FUNCTION_BLOCK E_CYCLE (* Peroidic event generator *)
  (* Standard: 61499-1 Annex A; Description: Copyright (c) 2017 fortiss GmbH This program and the accompanying materials are made available under the terms of the Eclipse Public License 2.0 which is available at https://www.eclipse.org/legal/epl-2.0/ SPDX-License-Identifier: EPL-2.0 *)
  (* Version 1.0, 2017-09-21, Alois Zoitl, fortiss GmbH, initial API and implementation and/or initial documentation *)
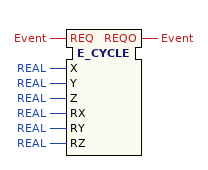
  EVENT_INPUT
    REQ; (* Move request *)
  END_EVENT
  EVENT_OUTPUT
    REQO; (* Move request output *)
  END_EVENT
  VAR_INPUT
    X : REAL; (* X value *)
    Y : REAL; (* Y value *)
    Z : REAL; (* Z value *)
    RX : REAL; (* RX value *)
    RY : REAL; (* RY value *)
    RZ : REAL; (* RZ value *)
  END_VAR
END_FUNCTION_BLOCK
